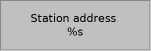
VISUALIZATION _VisuAddressShow  // 151x51
    Rectangle (1,1 148x48), "Station address %s", text variable: ComGVL._glAddressNameTable[ComGVL._glAddressSelectionIndex]
END_VISUALIZATION

(* stored: Version 1.1.0.1, ProductVersion 3.1.4024.2
   Visu _VisuAddressShow: Id {c266f1e4-b1ea-4287-b9b9-3ba0d597f098} *)
